Staubli VAL3: DeletePoint.pgx

program DeletePoint(num& bufferIn[])
  local string pointName
  local num i
begin
  //*******************************************************************************
  //*   ______
  //*  / _____) /|
  //* | |      / /
  //* | | /\  / /
  //* | | \ \/ /  _      Copyright (c) KEOLABS, 2016
  //* | |  \__/  | |        http://www.keolabs.com
  //* | |________| |
  //*  \__________/
  //*
  //********************************************************************************
  //*@file          : DeletePoint
  //*@author        : Yves Ragot
  //*@version       : $Id: DeletePoint.pgx 1198 2016-10-07 06:48:14Z yves $
  //*@brief         : Forget a memorized position point
  //*
  //*******************************************************************************/

  pointName = ""

  // get the name of the point
  for i = 0 to 9
      pointName = pointName + chr(bufferIn[17 + i])
  endFor

  if (len(pointName)) > 0

      // delete the point from the collection
      if (isDefined(pPointsTable[pointName]) == true)
          delete(pPointsTable[pointName])
      else
          GeneralStatus = 101
          LastErrorCode = 0
      endIf

  else
      GeneralStatus = 101
      LastErrorCode = 0
  endIf

end
